PROGRAM MAIN
VAR
END_VAR

END_PROGRAM

(* stored: Version 1.1.0.1
   POU MAIN: Id {2abaa063-5841-4cc9-93da-65614055800c} *)
